// TIA Portal V19 export
TYPE "LEXCHANGETRAY_typeSR1000Interface"
// configuration: LAF_typeSR1000Parameters
// commands: LEXCHANGETRAY_typeSR1000ManualCommands
// monitoring: LEXCHANGETRAY_typeSR1000ProcessValues
// stored: Access Published
   STRUCT
      configuration : "LAF_typeSR1000Parameters";
      commands { S7_SetPoint := 'True'} : "LEXCHANGETRAY_typeSR1000ManualCommands";
      monitoring { S7_SetPoint := 'True'} : "LEXCHANGETRAY_typeSR1000ProcessValues";
   END_STRUCT;
END_TYPE
